(*
Enables a FB to be registered in the Debug table for visibility within the IDE.  
Provides no additional functionality beyond this.
*)
INTERFACE I_Debug

END_INTERFACE

(* stored: Version 1.1.0.1
   Itf I_Debug: Id {dd9af94b-653d-4389-8fe6-660d00f8293a} *)
